{attribute 'qualified_only'}
VAR_GLOBAL CONSTANT
	ValueCountLimit : INT := 30;
	TableColumnLimit : INT := 10;
	
	BufferSize : INT := 1500;
	TableBufferSize : INT := 1000;
END_VAR

(* stored: Version 1.1.0.1
   GVL RecipeParameters: Id {d9be3204-2b08-0ff7-0d69-0af1093d67f3}, ParameterList True *)
